{attribute 'qualified_only'}
VAR_GLOBAL
	
 mb_Input_Coils    :    ARRAY [0..6] OF BOOL;
 mb_Output_Coils :    ARRAY [0..8] OF BOOL;
 Step_Index :   INT;
 
	nState: INT;
	nBoxCounter: INT;
END_VAR

(* stored: Version 1.1.0.1, ProductVersion 3.1.4024.12
   GVL GVL: Id {b2059115-329a-4a6a-9a68-32bdc03437c1} *)
